PROGRAM Singularity
VAR
	Inside_Dia: LREAL;
	At_Singularity: BOOL;
	Near_Singularity: BOOL;
	Singular_SimsX_Stop: MC_Stop;
	Singular_SimsY_Stop: MC_Stop;
	Singular_SimsZ_Stop: MC_Stop;
END_VAR

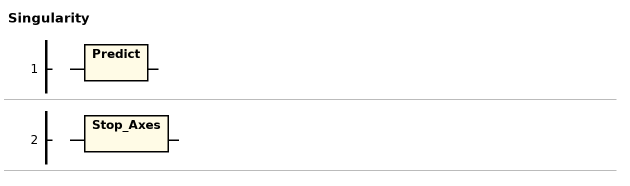
// NETWORK 1
Predict();

// NETWORK 2
Stop_Axes();

ACTION Predict:
Inside_Dia:= SQRT((SimsX.NcToPlc.ActPos)*(SimsX.NcToPlc.ActPos)+
				  (SimsY.NcToPlc.ActPos)*(SimsY.NcToPlc.ActPos));
		
IF Inside_Dia>=249 OR SimsZ.NcToPlc.ActPos>=65 OR SimsZ.NcToPlc.ActPos<=-155 THEN
	At_Singularity:=TRUE;
ELSE
	At_Singularity:=FALSE;	
END_IF

IF Inside_Dia>=240 OR SimsZ.NcToPlc.ActPos>=60 OR SimsZ.NcToPlc.ActPos<=-150 THEN
	Near_Singularity:=TRUE;
ELSE
	Near_Singularity:=FALSE;	
END_IF
END_ACTION

ACTION Reset:
// NETWORK 1
END_ACTION

ACTION Stop_Axes:
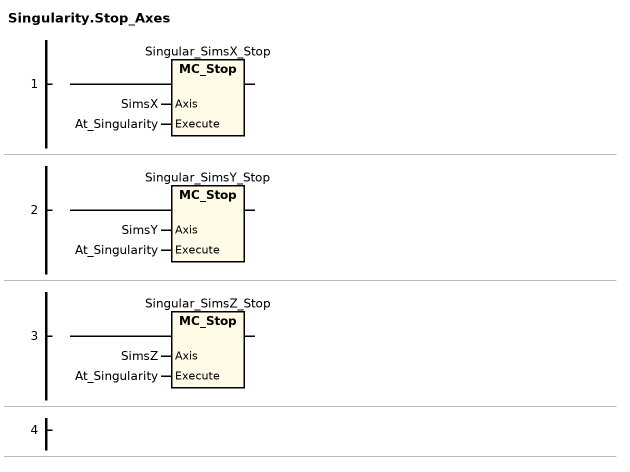
// NETWORK 1
Singular_SimsX_Stop(Axis := SimsX, Execute := At_Singularity); // MC_Stop

// NETWORK 2
Singular_SimsY_Stop(Axis := SimsY, Execute := At_Singularity); // MC_Stop

// NETWORK 3
Singular_SimsZ_Stop(Axis := SimsZ, Execute := At_Singularity); // MC_Stop

// NETWORK 4
END_ACTION

END_PROGRAM

(* stored: Version 1.1.0.1, ProductVersion 3.1.4018.9
   POU Singularity: Id {0e70836d-0845-4682-84ee-75e3692b8494}, SpecialFunc None
   Action Predict: Id {23a041e9-9765-4e8a-9727-aecf3f9e6314}
   Action Reset: Id {0591d492-dd86-4b22-b9e8-462e3698da70}
   Action Stop_Axes: Id {c2f4f3bc-375a-48ad-8b1e-ca921b9c7e12} *)
